{attribute 'GeneratedUsingTerminal: EK1561-0000-0018'}
{attribute addProperty BoxType "EK1561-0000-0018"}
{attribute addProperty Description "EK1561 1 port EtherCAT junction (POF)"}
{attribute addProperty Physics "K_KY"}
{attribute addProperty Id "InfoDataAT %I*InfoData_6F19DB2B2"}
{attribute addProperty CRC "532711307"}
{attribute addProperty Size "2"}
TYPE EK1561_1FC0878B EXTENDS EtcSlaveTerminalBase_947E5A46 :
STRUCT
	{attribute addProperty Name "InfoData"}
	InfoData : InfoData_6F19DB2B;
END_STRUCT
END_TYPE

(* stored: Version 1.2.0.0, ProductVersion 3.1.4024.9
   DUT EK1561_1FC0878B: Id {803f8a2b-4501-499c-97da-c4ad477b8ec0} *)
